// SIMATIC S7-200 project (STEP 7-Micro/WIN), CPU 222 REL 01.22

ORGANIZATION_BLOCK Main:OB1
TITLE=这个项目包含LY系列冷冻油专用滤油机控制模块，控制设备包括进油阀门、过滤泵、排油阀门和清洗泵。
// 
// 系统启动时，系统状态和批处理状态被清零，滤油机进入初始状态。
// 操作员按下启动按钮后，系统状态置为1，打开进油阀门，冷冻油开始流入滤油机。急停按钮用于在紧急情况下暂停系统操作。进油传感器检测到油液时，系统状态置为1，打开进油阀门，冷冻油开始流入滤油机。此时，进油定时器启动，确保进油时间可控。进油过程中，进油传感器持续检测，只有当其确认进油完成后，系统状态才会从1变为2，进入过滤阶段，否则系统保持等待，避免在无油情况下启动过滤。
// 进入过滤阶段后，程序调用过滤子程序，继续运行进油阀门，油液通过过滤器净化。过滤传感器监控过滤状态，若置位，则触发后续动作，同时进油定时器继续计时，确保过滤时间适当。当过滤完成且排油传感器未触发时，系统状态从2变为3，停止相关定时器，准备进入下一阶段。排油结束后，系统可进入清洗阶段，系统状态置为5，调用清理子程序，清空相关状态。此时，清洗泵根据内部信号启动，持续运行一段时间后关闭，确保清洗彻底。整个过程中，系统状态的转移按需逐步进行，从0到2，再到3、5，保证流程逻辑清晰。
// 此外，系统支持批处理功能，通过批处理主程序和批处理量判断程序控制。当批处理启用标志或启动按钮触发时，系统准备记录油量，目标值由流量预设值1和流量预设值2定义。一旦达到预设值，批处理指示灯1和批处理指示灯2更新状态，确保每次处理油量精确。流量计数器在批处理开始时复位，并在达到目标时触发中断，确保计数准确。
// 安全性是系统设计的核心。若急停按钮被按下，进油阀门、过滤泵、排油阀门和清洗泵必须立即关闭，防止意外运行。系统运行时，根据阶段独立工作，避免设备冲突。例如，在进油阶段优先运行进油阀门，过滤阶段优先运行过滤泵，确保各设备分工明确。
// 
BEGIN
Network 1 // 网络标题
// 网络注释
LD     SM0.1
MOVW   +0, VW0
AENO
MOVW   +0, VW2
Network 2
LDW=   VW0, +0
OW=    VW0, +4
OW=    VW0, +5
AN     M5.0
LDW=   VW0, +2
A      M4.0
LDW=   VW0, +3
A      M4.0
OLD
OLD
LPS
MOVW   +1, VW0
AENO
MOVB   1, MB2
LPP
CALL   ClearOutput:SBR5
Network 3
LD     I0.4
O      M4.1
AW=    VW0, +1
MOVW   +2, VW0
AENO
MOVB   2, MB2
AENO
MOVB   0, MB4
Network 4
LDN    I0.5
O      M4.2
AW=    VW0, +2
LPS
MOVW   +3, VW0
AENO
MOVB   4, MB2
AENO
R      T37, 2
LPP
MOVW   +0, VW22
AENO
MOVW   +0, VW24
AENO
MOVB   0, MB4
Network 5
LDW<=  VW0, +3
A      M5.0
LDW=   VW0, +4
AN     I0.5
OLD
LDW=   VW0, +4
AN     M3.6
OLD
LPS
MOVW   +5, VW0
AENO
MOVB   0, MB2
LPP
CALL   ClearOutput:SBR5
Network 6
LDW=   VW0, +5
A      M3.6
MOVW   +4, VW0
Network 7
LD     SM0.0
CALL   BatchMain:SBR3
Network 8
LDW=   VW0, +2
CALL   AutoFilter:SBR1
Network 9
LDW=   VW0, +3
CALL   AutoFilterNormalStop:SBR2
Network 10
LDW=   VW0, +4
CALL   HandleRun:SBR0
Network 11
LD     SM0.0
MOVW   VW10, VW4
AENO
*I     +10, VW4
AENO
MOVW   VW12, VW6
AENO
*I     +10, VW6
AENO
MOVW   VW14, VW8
*I     +10, VW8
Network 12
LDW<   VW0, +4
MOVB   0, MB3
END_ORGANIZATION_BLOCK

SUBROUTINE_BLOCK HandleRun:SBR0
TITLE=子程序注释
BEGIN
Network 1 // 网络标题
// 网络注释
LD     M3.0
=      Q0.0
TON    T37, VW4
Network 2
LD     Q0.0
A      Q0.2
A      T37
A      M3.1
=      Q0.1
Network 3
LD     M3.2
AN     I0.6
=      Q0.2
Network 4
LD     M3.3
A      T37
=      Q0.3
Network 5
LDN    M3.6
MOVB   0, MB3
END_SUBROUTINE_BLOCK

SUBROUTINE_BLOCK AutoFilter:SBR1
TITLE=
BEGIN
Network 1
LD     SM0.0
=      Q0.0
TON    T37, VW4
Network 4
LDN    I0.7
TON    T43, +50
Network 5
LD     T43
=      Q0.3
Network 6
LD     T37
A      Q0.0
A      Q0.2
=      Q0.1
Network 7
LD     I0.7
MOVW   +1, VW24
Network 8
LDW=   VW24, +1
=      Q0.2
Network 9
LD     I0.6
MOVW   +0, VW24
END_SUBROUTINE_BLOCK

SUBROUTINE_BLOCK AutoFilterNormalStop:SBR2
TITLE=
BEGIN
Network 1
LD     SM0.0
LPS
NOT
=      Q0.1
LPP
TON    T38, VW6
Network 2
LD     T38
R      Q0.0, 2
R      Q0.3, 2
Network 3
LDN    I0.6
TON    T39, VW8
Network 4
LD     T39
LPS
R      Q0.2, 2
MOVW   +0, VW0
AENO
R      T38, 2
LPP
R      T39, 2
END_SUBROUTINE_BLOCK

SUBROUTINE_BLOCK BatchMain:SBR3
TITLE=
BEGIN
Network 1
LD     M0.0
O      I0.3
AW=    VW2, +0
CALL   BatchVolumeJudge:SBR4
Network 2
LDW=   VW2, +1
A      M0.2
LPS
MOVW   +2, VW2
AENO
R      Q0.4, 2
R      Q0.5, 2
LPP
MOVB   12, SMB37
AENO
HSC    0
AENO
MOVB   4, MB1
Network 3
LDW=   VW2, +2
AN     M0.2
MOVB   0, MB0
AENO
MOVB   2, MB1
AENO
MOVW   +1, VW2
AENO
MOVB   140, SMB37
AENO
HSC    0
AENO
S      Q0.4, 1
S      Q0.5, 1
Network 4
LD     M0.1
MOVB   1, MB1
AENO
LDW=   VW2, +1
AW>=   VW26, VW28
MOVB   16, MB1
AENO
OLD
LPS
MOVB   0, MB0
AENO
MOVW   +0, VW2
AENO
R      Q0.4, 2
R      Q0.5, 2
LPP
LPS
MOVR   0.0, VD216
AENO
MOVR   0.0, VD220
AENO
MOVR   0.0, VD104
LPP
MOVB   12, SMB37
AENO
HSC    0
Network 5
LDW=   VW2, +1
LPS
DTR    HC0, VD208
AENO
ITD    VW16, VD212
AENO
DTR    VD212, VD212
LPP
MOVR   VD208, VD112
AENO
/R     VD212, VD112
AENO
*R     1000.0, VD112
AENO
DTI    HC0, VW18
Network 6
LDW=   VW2, +1
LPS
AN     T40
TON    T40, +10
LPP
MOVW   C0, VW26
Network 7
LD     T40
LPS
MOVR   VD220, VD216
AENO
MOVR   VD112, VD220
AENO
MOVR   VD220, VD104
-R     VD216, VD104
LPP
+R     VD104, VD136
AENO
+R     VD104, VD140
Network 8
LD     T40
LDW=   VW2, +0
CTU    C0, +32767
Network 9
LD     M1.4
TON    T41, +50
Network 10
LD     M1.3
TON    T42, +50
Network 11
LD     T41
O      T42
MOVB   1, MB1
Network 12
LDW=   VW2, +0
LPS
A      M20.0
MOVR   0.0, VD136
AENO
MOVR   0.0, VD140
AENO
R      M20.0, 2
LRD
A      M20.1
MOVR   0.0, VD140
AENO
R      M20.1, 2
LRD
AR>=   VD136, 100000000.0
MOVR   0.0, VD136
AENO
MOVR   0.0, VD140
LPP
AR>=   VD140, 100000000.0
MOVR   0.0, VD140
END_SUBROUTINE_BLOCK

SUBROUTINE_BLOCK BatchVolumeJudge:SBR4
TITLE=
BEGIN
Network 1
LD     SM0.0
LPS
ITD    VW16, VD212
AENO
DTR    VD212, VD212
AENO
/R     1000.0, VD212
LRD
*R     VD108, VD212
AENO
*R     VD100, VD212
AENO
ROUND  VD212, VD124
LRD
MOVR   VD108, VD212
AENO
/R     VD80, VD212
AENO
ROUND  VD212, VD212
LPP
DTI    VD212, VW20
AENO
MOVW   +3, VW28
AENO
*I     VW20, VW28
AENO
MOVW   +0, VW26
Network 2
LD     SM0.0
LPS
ITD    VW16, VD212
AENO
DTR    VD212, VD212
LPP
/R     1000.0, VD212
AENO
*R     VD116, VD212
AENO
ROUND  VD212, VD128
Network 3
LD     SM0.0
LPS
ITD    VW16, VD212
AENO
DTR    VD212, VD212
LPP
/R     1000.0, VD212
AENO
*R     VD120, VD212
AENO
ROUND  VD212, VD132
Network 4
LD     SM0.0
MOVD   VD124, VD200
AENO
-D     VD128, VD200
AENO
MOVD   VD124, VD204
-D     VD132, VD204
Network 5
LD     SM0.0
LPS
MOVD   +0, SMD38
AENO
MOVD   VD200, SMD42
AENO
MOVB   236, SMB37
AENO
HDEF   0, 1
LRD
ATCH   BatchArrive:INT0, 12
AENO
ENI
LPP
HSC    0
Network 6
LD     SM0.0
LPS
MOVB   0, MB0
AENO
MOVB   2, MB1
AENO
MOVW   +1, VW2
AENO
=      Q0.4
=      Q0.5
LPP
MOVR   0.0, VD216
AENO
MOVR   0.0, VD216
Network 7
LD     SM0.0
MOVR   VD136, VD144
AENO
MOVR   VD140, VD148
END_SUBROUTINE_BLOCK

SUBROUTINE_BLOCK ClearOutput:SBR5
TITLE=
BEGIN
Network 1
LD     SM0.0
LPS
MOVB   0, MB3
AENO
=      L63.7
LRD
MOVW   +0, VW22
AENO
O      L63.7
=      L63.6
LRD
MOVW   +0, VW24
AENO
O      L63.6
=      L63.5
LPP
MOVB   0, MB4
AENO
O      L63.5
R      Q0.0, 2
R      Q0.3, 2
R      Q0.4, 2
R      M3.6, 0
R      T37, 2
R      T38, 2
R      T39, 2
R      Q0.1, 2
END_SUBROUTINE_BLOCK

INTERRUPT_BLOCK BatchArrive:INT0
TITLE=中断程序注释
BEGIN
Network 1 // 网络标题
// 网络注释
LDD>=  HC0, VD200
MOVB   172, SMB37
AENO
MOVD   VD204, SMD42
AENO
HSC    0
AENO
R      Q0.5, 2
Network 2
LDD>=  HC0, VD204
LPS
MOVW   +0, VW2
AENO
MOVB   8, MB1
AENO
MOVB   12, SMB37
AENO
HSC    0
AENO
R      Q0.4, 2
LRD
MOVR   0.0, VD104
AENO
MOVR   0.0, VD216
AENO
MOVR   0.0, VD220
LPP
MOVR   VD144, VD136
AENO
+R     VD112, VD136
AENO
MOVR   VD148, VD140
+R     VD112, VD140
END_INTERRUPT_BLOCK

DATA_BLOCK_TAB USER1
BEGIN
VW0      0
VW2      0
VW10     5
VW12     60
VW14     10
VW16     7282
VW18     0
VW20     0
VD80     5.0
VD100    1.0
VD104    0.0
VD108    1000.0
VD112    0.0
VD116    0.0
VD120    0.0
VD124    10200
VD128    0
VD132    0
END_DATA_BLOCK_TAB
